
FUNCTION CB_real_to_dword : DWORD

TITLE = ' Convert a real into an integer '
VERSION : '1.0'
AUTHOR  : CB
NAME    : realDwor
FAMILY  : TNI

VAR_INPUT
    IN : REAL;
END_VAR

VAR_TEMP

END_VAR

BEGIN

CB_real_to_dword := DINT_TO_DWORD(REAL_TO_DINT(IN));

END_FUNCTION
